// TwinCAT 3 PLC project MachineControl
// Title: Tk_MachineControl
// Company: Komatsu
// Author: TK
// ProjectVersion: 0.0.3.1
// Description: マシンの管理用ライブラリ アラーム、4024用イベントリード、マシンステート
// ProgramVersion: 3.1.4026.26
// libraries:
//   Tc2_Standard, * (Beckhoff Automation GmbH)
//   Tc2_System, * (Beckhoff Automation GmbH)
//   Tc2_Utilities, * (Beckhoff Automation GmbH)
//   Tc3_EventLogger, * (Beckhoff Automation GmbH)
// project tree:
//   Alarm/ FB_Alarm.TcPOU (not stored), FB_AlarmFromTcMessage.TcPOU (not stored)
//   EventRead/ FB_EventListener.TcPOU (not stored), ST_EventRead.TcDUT (not stored)
//   MachineState/ FB_MachineState_Sample.TcPOU (not stored)
//   MachineState/Original/ E_MachineState.TcDUT (not stored), FB_MachineState.TcPOU (not stored)
//   MachineState/Ref PackML/ E_PackMLCommand.TcDUT, E_PackMLState.TcDUT, E_PackMLUnitMode.TcDUT (not stored), FB_PackMLStateMachine.TcPOU (not stored), FB_PackMLUnitModeManager.TcPOU (not stored), ST_PMLSubUnitInfo.TcDUT
//   Version/ Global_Version.TcGVL
// (motion and I/O tree: see PLC project wago7871664000080)
// real-time tasks:
//   TASK PlcTask: cycle T#10ms, priority 20, ADS port 350

// ---- MachineState/Ref PackML/E_PackMLCommand.TcDUT
{attribute 'qualified_only'}
{attribute 'strict'}
{attribute 'to_string'}
TYPE E_PackMLCommand :
(
    Undefined   := 0,
    Reset       := 1,
    Start       := 2,
    Stop        := 3,
    Hold        := 4,
    Unhold      := 5,
    Suspend		:= 6,
    Unsuspend	:= 7,
    Abort       := 8,
    Clear       := 9,
    Complete    := 10
);
END_TYPE

// ---- MachineState/Ref PackML/E_PackMLState.TcDUT
{attribute 'qualified_only'}
{attribute 'strict'}
{attribute 'to_string'}
TYPE E_PackMLState : 
(
	Undefined		:= 0,
	Clearing		:= 1,		//Clearing（異常解除中）		Acting	Abort後の異常解除およびStopped状態への移行中
	Stopped			:= 2,		//Stopped（停止）				Wait	制御された停止状態、再開にはリセット（Reset）が必要
	Starting		:= 3,		//Starting（開始中）			Acting	生産に向けて稼働を立ち上げ中
	Idle			:= 4,		//Idle（待機）					Wait	開始準備完了、開始（Start）指令待ち
	Suspended		:= 5,		//Suspended（中断）				Wait	外部要因（上流・下流工程など）による一時停止
	Execute			:= 6,		//Execute（実行中）				Acting	生産中（稼働状態）
	Stopping		:= 7,		//Stopping（停止処理中）		Acting	制御された減速による停止（Stopped）への移行
	Aborting		:= 8,		//Aborting（異常停止中）		Acting	緊急停止シーケンスの実行中
	Aborted			:= 9,		//Aborted（異常停止）			Wait	異常状態、異常の解消とリセット（Reset）が必要
	Holding			:= 10,		//Holding（一時停止中）			Acting	Held状態へ移行中
	Held			:= 11,		//Held（一時停止）				Wait	オペレーターによる一時停止
	Unholding		:= 12,		//Unholding（一時停止解除中）	Acting	Held状態からExecute状態へ復帰中
	Suspending		:= 13,		//Suspending（中断中）			Acting	外部要因によりSuspended状態へ移行中
	Unsuspending	:= 14,		//Unsuspending（中断解除中）	Acting	Suspended状態からExecute状態へ復帰中
	Resetting		:= 15,		//Resetting（リセット中）		Acting	Idle状態への復帰準備中
	Completing		:= 16,		//Completing（完了処理中）		Acting	現在の生産サイクルを終了中
	Completed		:= 17		//Complete（完了）				Wait	サイクル終了、リセット（Reset）待ち
);
END_TYPE

// ---- MachineState/Ref PackML/ST_PMLSubUnitInfo.TcDUT
TYPE ST_PMLSubUnitInfo :
STRUCT
    bActive  : BOOL;
    eState   : E_PackMLState;
END_STRUCT
END_TYPE

// ---- Version/Global_Version.TcGVL
{attribute 'TcGenerated'}
{attribute 'no-analysis'}
{attribute 'linkalways'}
// This function has been automatically generated from the project information.
VAR_GLOBAL CONSTANT
	{attribute 'const_non_replaced'}
	stLibVersion_Tk_MachineControl : ST_LibVersion := (iMajor := 0, iMinor := 0, iBuild := 3, iRevision := 1, nFlags := 0, sVersion := '0.0.3.1');
END_VAR
